FUNCTION_BLOCK FB_DataCollectionSequence_Test EXTENDS FB_TestSuite
VAR
END_VAR


GivenThatSystemIsNotCalibratedDontAllowToStartSequence();


METHOD PRIVATE GivenThatSystemIsNotCalibratedDontAllowToStartSequence
VAR
    fbSystemCalibrationTestDouble : FB_SystemCalibrationTestDouble;
    fbResetSequenceTestDouble : FB_ResetSequenceTestDouble;
    fbTriggerManagerTestDouble : FB_TriggerManagerTestDouble;
    fbDataCollectionSequence : FB_DataCollectionSequence(iSystemCalibration := fbSystemCalibrationTestDouble,
                                                         iResetSequence := fbResetSequenceTestDouble,
                                                         iTriggerManager := fbTriggerManagerTestDouble);

    bErrorReturn : BOOL;
    sErrorStringReturn : T_MaxString;
END_VAR

TEST(__POUNAME());

fbResetSequenceTestDouble.SetIsReset(bIsReset := TRUE);
fbSystemCalibrationTestDouble.SetIsCalibrated(bIsCalibrated := FALSE);


fbDataCollectionSequence.Start(bError => bErrorReturn,
                               sErrorString => sErrorStringReturn);

AssertTrue(Condition := bErrorReturn,
           Message := 'Expected error');

AssertTrue(Condition := sErrorStringReturn <> '',
           Message := 'Expected non-empty string');

TEST_FINISHED();
END_METHOD

END_FUNCTION_BLOCK

(* stored: Version 1.1.0.1
   POU FB_DataCollectionSequence_Test: Id {ac62226e-fce3-4951-ba37-0043fdbb4f06}, SpecialFunc None
   Method GivenThatSystemIsNotCalibratedDontAllowToStartSequence: Id {50d7a577-1f67-4c0c-acd7-565fdd628fc8} *)
